{attribute 'GeneratedUsingTerminal: EL6021-0000-0018'}
{attribute addProperty BoxType "EL6021-0000-0018"}
{attribute addProperty Id "EtcSlaveTerminalBaseCOM_TxPDO_Map_InputsAT %I*COM_TxPDO_Map_Inputs_3801C95E30COM_RxPDO_Map_OutputsAT %Q*COM_RxPDO_Map_Outputs_DEF408EC27WcStateAT %I*WcState_9091E0EB2InfoDataAT %I*InfoData_32EB74EA10"}
{attribute addProperty CRC "2185377966"}
{attribute addProperty Size "69"}
TYPE EL6021_824238AE EXTENDS EtcSlaveTerminalBase :
STRUCT
	{attribute addProperty Name "COM_TxPDO_Map_Inputs"}
	COM_TxPDO_Map_Inputs : COM_TxPDO_Map_Inputs_3801C95E;
	{attribute addProperty Name "COM_RxPDO_Map_Outputs"}
	COM_RxPDO_Map_Outputs : COM_RxPDO_Map_Outputs_DEF408EC;
	{attribute addProperty Name "WcState"}
	WcState : WcState_9091E0EB;
	{attribute addProperty Name "InfoData"}
	InfoData : InfoData_32EB74EA;
END_STRUCT
END_TYPE

(* stored: Version 1.2.0.0, ProductVersion 3.1.4024.9
   DUT EL6021_824238AE: Id {6d51cb24-c1fb-491b-bcb1-19f9df65299d} *)
